Fanuc KAREL source: UNINIT.kl

PROGRAM T
%NOLOCKGROUP
VAR
 v0 : REAL
 res : BOOLEAN
BEGIN
 res = UNINIT(v0)
END T
